(* PLC project SafeLOGIC-1, BrAutomation SafeDESIGNER  4.3.4.4 *)
(* stored: companyURL http://www.br-automation.com, creationDateTime Thu Jun 24 15:49:10 2021 *)

PROGRAM Main
  VAR  (* added by the conversion: wires and edge detectors of the diagram *)
    _SAFEBOOL_TO_BOOL19_OUT : BOOL;
  END_VAR

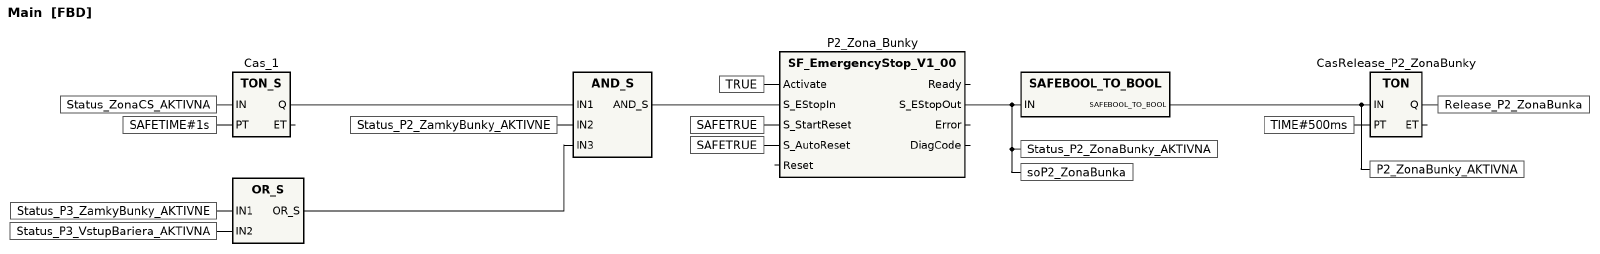
(* FBD diagram, written out as Structured Text *)
Cas_1(IN := Status_ZonaCS_AKTIVNA, PT := SAFETIME#1s);
P2_Zona_Bunky(Activate := TRUE, S_EStopIn := AND_S(Cas_1.Q, Status_P2_ZamkyBunky_AKTIVNE, OR_S(Status_P3_ZamkyBunky_AKTIVNE, Status_P3_VstupBariera_AKTIVNA)), S_StartReset := SAFETRUE, S_AutoReset := SAFETRUE);
Status_P2_ZonaBunky_AKTIVNA := P2_Zona_Bunky.S_EStopOut;
soP2_ZonaBunka := P2_Zona_Bunky.S_EStopOut;
_SAFEBOOL_TO_BOOL19_OUT := SAFEBOOL_TO_BOOL(P2_Zona_Bunky.S_EStopOut);
P2_ZonaBunky_AKTIVNA := _SAFEBOOL_TO_BOOL19_OUT;
CasRelease_P2_ZonaBunky(IN := _SAFEBOOL_TO_BOOL19_OUT, PT := TIME#500ms);
Release_P2_ZonaBunka := CasRelease_P2_ZonaBunky.Q;
END_PROGRAM
